FUNCTION_BLOCK PICKER_MODEL_CENTRAL (* Composite Function Block Type *)
  (* Standard: 61499-2 *)
  (* Version 0.2, 2003-12-05, JHC, Rockwell Automation, Renamed from NEWCOMPFB. *)
  (* Version 0.1, 2002-01-08, JHC, Rockwell Automation, Added DLY FB as example. *)
  (* Version 0.0, 2000-05-27, JHC, Rockwell Automation *)
  (* Compiler header: package fb.rt.pnp; *)
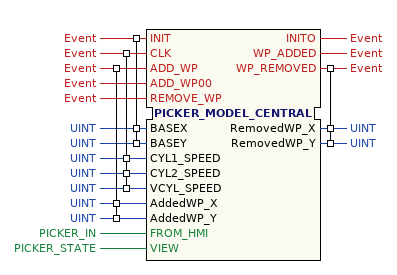
  EVENT_INPUT
    INIT WITH BASEX, BASEY; (* Initialisation *)
    CLK WITH CYL1_SPEED, CYL2_SPEED, VCYL_SPEED;
    ADD_WP WITH AddedWP_X, AddedWP_Y;
    ADD_WP00;
    REMOVE_WP;
  END_EVENT
  EVENT_OUTPUT
    INITO; (* Initialization Confirm *)
    WP_ADDED;
    WP_REMOVED WITH RemovedWP_X, RemovedWP_Y;
  END_EVENT
  VAR_INPUT
    BASEX : UINT;
    BASEY : UINT;
    CYL1_SPEED : UINT;
    CYL2_SPEED : UINT;
    VCYL_SPEED : UINT;
    AddedWP_X : UINT;
    AddedWP_Y : UINT;
  END_VAR
  VAR_OUTPUT
    RemovedWP_X : UINT;
    RemovedWP_Y : UINT;
  END_VAR
  SOCKETS
    FROM_HMI : PICKER_IN;
    VIEW : PICKER_STATE;
  END_SOCKETS
  FBS
    MODEL : Model;
    CONTROL : CentralizedControl;
  END_FBS
  EVENT_CONNECTIONS
    INIT TO MODEL.INIT;
    MODEL.INITO TO VIEW.INIT;
    CLK TO MODEL.CLK;
    ADD_WP TO MODEL.ADD_WP;
    REMOVE_WP TO MODEL.REMOVE_WP;
    MODEL.WP_ADDED TO WP_ADDED;
    MODEL.WP_REMOVED TO WP_REMOVED;
    ADD_WP00 TO MODEL.ADD_WP00;
    MODEL.CNF TO VIEW.CHG;
    FROM_HMI.REQ TO MODEL.REQ;
    MODEL.INITO TO CONTROL.INIT;
    MODEL.CHG TO CONTROL.REQ;
    CONTROL.INITO TO INITO;
    CONTROL.CNF TO MODEL.CYL_IND;
  END_CONNECTIONS
  DATA_CONNECTIONS
    MODEL.BASE_X TO VIEW.BASE_X;
    MODEL.BASE_Y TO VIEW.BASE_Y;
    MODEL.CYL1_X TO VIEW.CYL1_X;
    MODEL.CYL1_Y TO VIEW.CYL1_Y;
    MODEL.CYL2_X TO VIEW.CYL2_X;
    MODEL.CYL2_Y TO VIEW.CYL2_Y;
    MODEL.VCYL_X TO VIEW.VCYL_X;
    MODEL.VCYL_Y TO VIEW.VCYL_Y;
    MODEL.WP_X TO VIEW.WP1_X;
    MODEL.WP_Y TO VIEW.WP1_Y;
    MODEL.VACUUM_ON TO VIEW.VACUUM_ON;
    BASEX TO MODEL.BASEX;
    BASEY TO MODEL.BASEY;
    CYL1_SPEED TO MODEL.CYL1_SPEED;
    CYL2_SPEED TO MODEL.CYL2_SPEED;
    VCYL_SPEED TO MODEL.VCYL_SPEED;
    AddedWP_X TO MODEL.AddedWP_X;
    AddedWP_Y TO MODEL.AddedWP_Y;
    MODEL.RemovedWP_X TO RemovedWP_X;
    MODEL.RemovedWP_Y TO RemovedWP_Y;
    MODEL.WP3_X TO VIEW.WP3_X;
    MODEL.WP3_Y TO VIEW.WP3_Y;
    MODEL.WP2_X TO VIEW.WP2_X;
    MODEL.WP2_Y TO VIEW.WP2_Y;
    FROM_HMI.add1 TO MODEL.Add1;
    FROM_HMI.add2 TO MODEL.Add2;
    FROM_HMI.add3 TO MODEL.Add3;
    MODEL.c1home TO CONTROL.c1Home;
    MODEL.c1end TO CONTROL.c1End;
    MODEL.c2home TO CONTROL.c2Home;
    MODEL.c2end TO CONTROL.c2End;
    MODEL.vchome TO CONTROL.vcHome;
    MODEL.vcend TO CONTROL.vcEnd;
    MODEL.VACUUM_ON TO CONTROL.vac;
    CONTROL.vcExtend TO MODEL.vcyl_down;
    CONTROL.vacuum_on TO MODEL.vacuum_on;
    CONTROL.c1Extend TO MODEL.cyl1_fwd;
    CONTROL.c1Retract TO MODEL.cyl1_back;
    CONTROL.c2Extend TO MODEL.cyl2_fwd;
    CONTROL.c2Retract TO MODEL.cyl2_back;
    MODEL.pp1 TO CONTROL.pp1;
    MODEL.pp2 TO CONTROL.pp2;
    MODEL.pp3 TO CONTROL.pp3;
    CONTROL.vacuum_off TO MODEL.vacuum_off;
  END_CONNECTIONS
END_FUNCTION_BLOCK
